ABB RAPID module: Wizard.modx

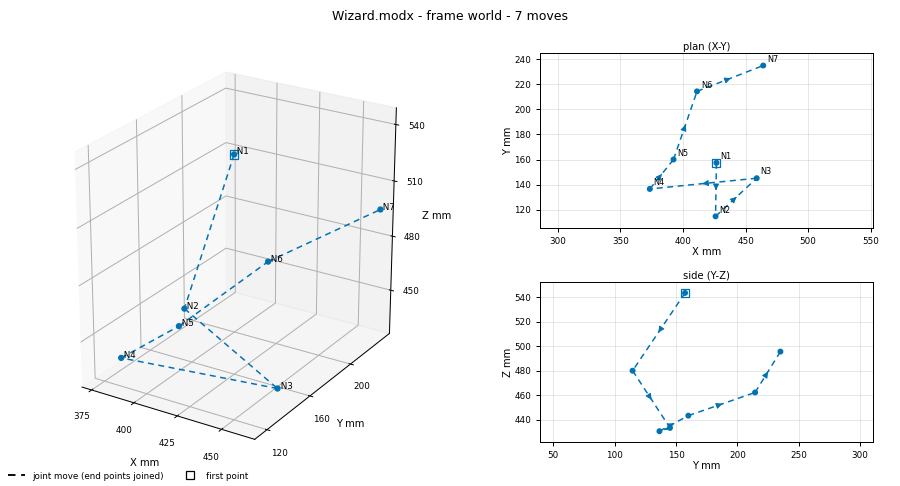
[picture p0: tool path of Wizard.modx in frame world, 7 of 7 moves have a stored position in this frame; points joined in program order, loops and branches not executed]
MODULE Wizard
PERS robtarget L1:=[[458.896423339844, 258.018341064453, 499.168701171875], [0.158319264650345, -0.310999274253845, -0.906924486160278, -0.236013606190681], [0, 0, 0, 0], [9000000000, 9000000000, 9000000000, 9000000000, 9000000000, 9000000000]];
PERS robtarget L2:=[[453.003936767578, 238.157562255859, 498.891326904297], [0.173174694180489, -0.318663984537125, -0.903377771377563, -0.228850185871124], [0, 0, 0, 0], [9000000000, 9000000000, 9000000000, 9000000000, 9000000000, 9000000000]];
PERS robtarget L3:=[[467.207946777344, 257.174133300781, 502.668334960938], [0.188314989209175, -0.247268840670586, -0.942852318286896, -0.12010432779789], [0, 0, 0, 0], [9000000000, 9000000000, 9000000000, 9000000000, 9000000000, 9000000000]];
PERS robtarget L4:=[[514.964782714844, 218.257675170898, 489.758850097656], [0.254175692796707, 0.157829031348228, -0.943383932113647, -0.143218100070953], [0, 0, -1, 0], [9000000000, 9000000000, 9000000000, 9000000000, 9000000000, 9000000000]];
PERS robtarget L5:=[[547.214965820313, 290.206146240234, 497.397125244141], [0.288632273674011, 0.230073392391205, -0.926952660083771, -0.067203991115093], [0, 0, -1, 0], [9000000000, 9000000000, 9000000000, 9000000000, 9000000000, 9000000000]];
PERS robtarget L6:=[[527.039978027344, 356.929534912109, 494.073699951172], [0.316573202610016, 0.293845564126968, -0.901871979236603, 0.00794433057308197], [0, 0, -1, 0], [9000000000, 9000000000, 9000000000, 9000000000, 9000000000, 9000000000]];
PERS robtarget M1:=[[236.863128662109, 297.165222167969, 440.828704833984], [0.32827416062355, -0.426665514707565, -0.742763459682465, -0.398114413022995], [0, 0, 0, 0], [9000000000, 9000000000, 9000000000, 9000000000, 9000000000, 9000000000]];
PERS robtarget M2:=[[218.475021362305, 287.130126953125, 464.338653564453], [0.296256810426712, -0.342145889997482, -0.805417358875275, -0.382715255022049], [0, 0, 0, 0], [9000000000, 9000000000, 9000000000, 9000000000, 9000000000, 9000000000]];
PERS robtarget M3:=[[179.02392578125, 353.076507568359, 493.904052734375], [0.115374229848385, -0.0449087247252464, -0.969848573207855, -0.209918528795242], [0, 0, 0, 0], [9000000000, 9000000000, 9000000000, 9000000000, 9000000000, 9000000000]];
PERS robtarget M4:=[[144.812072753906, 402.534454345703, 487.075408935547], [0.0055272919125855, -0.133435189723969, 0.985181629657745, 0.107618115842342], [0, 0, 0, 0], [9000000000, 9000000000, 9000000000, 9000000000, 9000000000, 9000000000]];
PERS robtarget M5:=[[122.549194335938, 425.369964599609, 477.968231201172], [0.0256542544811964, -0.173865929245949, 0.977084934711456, 0.120072849094868], [0, 0, 0, 0], [9000000000, 9000000000, 9000000000, 9000000000, 9000000000, 9000000000]];
PERS robtarget M6:=[[244.420532226563, 276.978149414063, 405.151458740234], [0.406883299350739, -0.511724472045898, -0.634383738040924, -0.412481904029846], [0, 1, 0, 0], [9000000000, 9000000000, 9000000000, 9000000000, 9000000000, 9000000000]];
PERS robtarget N1:=[[426.733428955078, 157.378616333008, 543.441040039063], [0.123705096542835, -0.544608473777771, -0.675274968147278, -0.481770038604736], [0, 0, 0, 0], [9000000000, 9000000000, 9000000000, 9000000000, 9000000000, 9000000000]];
PERS robtarget N2:=[[426.039581298828, 114.640037536621, 480.103149414063], [0.079576939344406, -0.562970638275146, -0.723652005195618, -0.39122799038887], [0, 0, 0, 0], [9000000000, 9000000000, 9000000000, 9000000000, 9000000000, 9000000000]];
PERS robtarget N3:=[[458.906677246094, 145.095626831055, 433.575286865234], [0.125698193907738, -0.708085536956787, -0.51935076713562, -0.461616307497025], [0, 1, 0, 0], [9000000000, 9000000000, 9000000000, 9000000000, 9000000000, 9000000000]];
PERS robtarget N4:=[[373.535797119141, 136.527557373047, 430.798614501953], [0.183426380157471, -0.798300683498383, -0.27296394109726, -0.504540860652924], [0, 1, 0, 0], [9000000000, 9000000000, 9000000000, 9000000000, 9000000000, 9000000000]];
PERS robtarget N5:=[[392.482513427734, 160.054794311523, 443.464935302734], [0.078961528837681, -0.68575531244278, -0.554902672767639, -0.464314341545105], [0, 0, 0, 0], [9000000000, 9000000000, 9000000000, 9000000000, 9000000000, 9000000000]];
PERS robtarget N6:=[[411.233276367188, 214.447677612305, 462.356842041016], [0.0290174279361963, -0.799260258674622, -0.390972465276718, -0.455501466989517], [0, 1, 0, 1], [9000000000, 9000000000, 9000000000, 9000000000, 9000000000, 9000000000]];
PERS robtarget N7:=[[464.075408935547, 235.073638916016, 495.652740478516], [0.125889465212822, 0.980195045471191, -0.0606890581548214, 0.140308231115341], [0, 1, 0, 1], [9000000000, 9000000000, 9000000000, 9000000000, 9000000000, 9000000000]];
PERS robtarget P5:=[[662.454223632813, 306.828918457031, 567.975402832031], [0.470702201128006, -0.07366531342268, -0.878970563411713, -0.0205820631235838], [0, 0, 0, 0], [9000000000, 9000000000, 9000000000, 9000000000, 9000000000, 9000000000]];
PERS robtarget P6:=[[620.727355957031, 374.223602294922, 520.497192382813], [0.530443906784058, -0.0285077802836895, -0.847173392772675, 0.010668414644897], [0, 0, 0, 0], [9000000000, 9000000000, 9000000000, 9000000000, 9000000000, 9000000000]];
PERS robtarget P7:=[[631.871276855469, 348.450347900391, 478.40869140625], [0.473697394132614, -0.075770862400532, -0.870681822299957, 0.108548432588577], [0, 0, 0, 0], [9000000000, 9000000000, 9000000000, 9000000000, 9000000000, 9000000000]];
PERS robtarget Pierko1:=[[661.21337890625, 279.395416259766, 637.873046875], [0.525981545448303, -0.07453079521656, -0.834759771823883, -0.144791930913925], [0, 0, 0, 0], [9000000000, 9000000000, 9000000000, 9000000000, 9000000000, 9000000000]];
PERS robtarget Pierko2:=[[696.242004394531, 258.929077148438, 600.872741699219], [0.485446214675903, 0.0299419183284044, -0.846789836883545, -0.215389013290405], [0, 0, 0, 0], [9000000000, 9000000000, 9000000000, 9000000000, 9000000000, 9000000000]];
PERS robtarget Pierko3:=[[661.213073730469, 279.395751953125, 637.87255859375], [0.525982856750488, -0.074529871344566, -0.834758996963501, -0.144792139530182], [0, 0, 0, 0], [9000000000, 9000000000, 9000000000, 9000000000, 9000000000, 9000000000]];
PERS robtarget Pierko4:=[[656.249267578125, 281.760528564453, 600.59912109375], [0.533924996852875, -0.0333066247403622, -0.84251993894577, -0.063047096133232], [0, 0, 0, 0], [9000000000, 9000000000, 9000000000, 9000000000, 9000000000, 9000000000]];
	PROC main()
MoveJ N1, v1000, fine, tool0;
MoveJ N2, v1000, fine, tool0;
MoveJ N3, v1000, fine, tool0;
MoveJ N4, v1000, fine, tool0;
MoveJ N5, v1000, fine, tool0;
MoveJ N6, v1000, fine, tool0;
MoveJ N7, v1000, fine, tool0;
	ENDPROC
ENDMODULE
